FUNCTION_BLOCK Relay
VAR
	bOutput	AT%Q*	: BOOL;
	tonPulse		: TON;
	tonPulseAcyclic	: TON;
END_VAR

// tonPulseAcyclic();
// 
// IF tonPulseAcyclic.Q THEN
// 	SwitchOff();
// 	tonPulseAcyclic(IN := FALSE);
// END_IF

METHOD Cyclic
VAR_INPUT
END_VAR
tonPulseAcyclic();

IF tonPulseAcyclic.Q THEN
	SwitchOff();
	tonPulseAcyclic(IN := FALSE);
END_IF
END_METHOD

METHOD Pulse : BOOL
VAR_INPUT
	tPulseTime	: TIME;
END_VAR
tonPulse(IN := TRUE, PT:= tPulseTime);

IF NOT tonPulse.Q THEN
	SwitchOn();
ELSIF tonPulse.Q THEN
	SwitchOff();
	tonPulse(IN := FALSE);
	Pulse := TRUE;
END_IF
END_METHOD

METHOD PulseAcyclic : BOOL
VAR_INPUT
	tPulseTime	: TIME;
END_VAR
SwitchOn();
tonPulseAcyclic.IN := TRUE;
tonPulseAcyclic.PT := tPulseTime;

PulseAcyclic := TRUE;
END_METHOD

PROPERTY State : BOOL
GET
State := bOutput;
END_GET
END_PROPERTY

METHOD SwitchOff : BOOL
VAR_INPUT
END_VAR
bOutput := FALSE;

SwitchOff := TRUE;
END_METHOD

METHOD SwitchOn : BOOL
VAR_INPUT
END_VAR
bOutput := TRUE;

SwitchOn := TRUE;
END_METHOD

END_FUNCTION_BLOCK

(* stored: Version 1.1.0.1
   POU Relay: Id {5085b1cf-4d06-4906-8007-1329dfffaf0f}, SpecialFunc None
   Method Cyclic: Id {224f8fb9-8aec-44dd-a993-3e3002545e72}
   Method Pulse: Id {1937db57-4c05-4d40-92ff-67b59d714bee}
   Method PulseAcyclic: Id {890da05d-c0eb-4dfb-98d9-20ced296544c}
   Property State: Id {50ff1f51-76e6-4379-a499-b34c966063f1}
   Get Get: Id {c074bbf0-f69b-4bd3-a56c-637e0627ed6f}
   Method SwitchOff: Id {71d54ee8-6e93-447d-8209-bf17b3119904}
   Method SwitchOn: Id {c87da857-2505-48e7-b65d-b923003a41ae} *)
